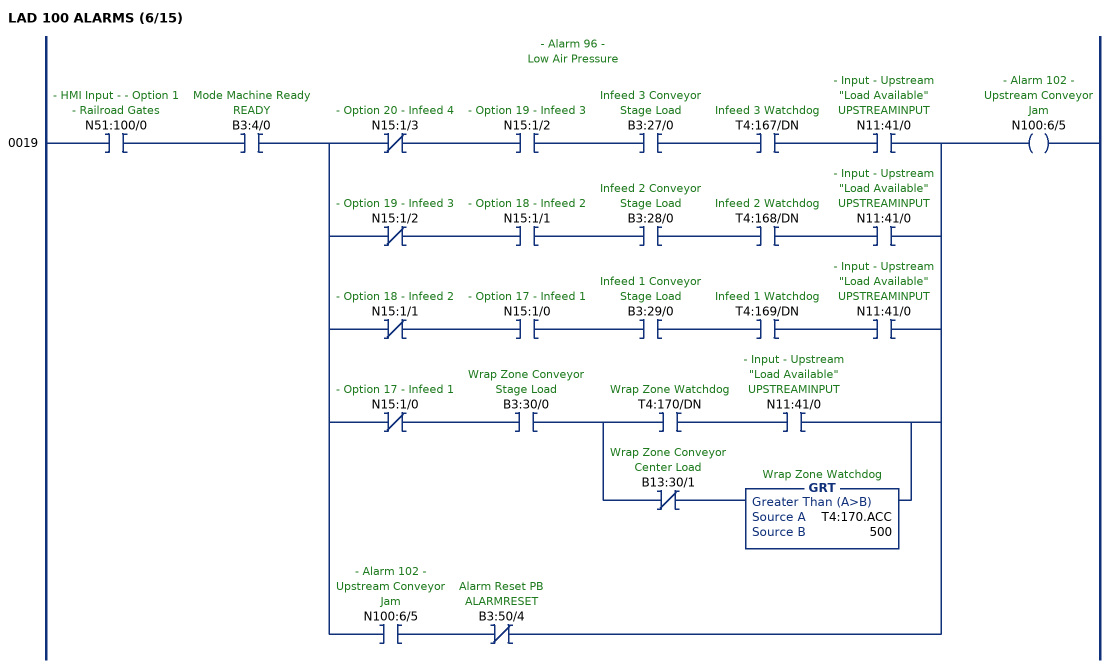
% Rung: 19 %
% - Alarm 96 -
% 
% Low Air Pressure %
SOR XIC N51:100/0 XIC B3:4/0 BST XIO N15:1/3 XIC N15:1/2 XIC B3:27/0 XIC T4:167/DN XIC N11:41/0 NXB XIO N15:1/2 XIC N15:1/1 XIC B3:28/0 XIC T4:168/DN XIC N11:41/0 NXB XIO N15:1/1 XIC N15:1/0 XIC B3:29/0 XIC T4:169/DN XIC N11:41/0 NXB XIO N15:1/0 XIC B3:30/0 BST XIC T4:170/DN XIC N11:41/0 NXB XIO B13:30/1 GRT T4:170.ACC 500 BND NXB XIC N100:6/5 XIO B3:50/4 BND OTE N100:6/5 EOR
%   N51:100/0  "- HMI Input - - Option 1 - Railroad Gates" %
%   B3:4/0  READY  "Mode Machine Ready" %
%   N15:1/3  "- Option 20 - Infeed 4" %
%   N15:1/2  "- Option 19 - Infeed 3" %
%   B3:27/0  "Infeed 3 Conveyor Stage Load" %
%   T4:167  "Infeed 3 Watchdog" %
%   N11:41/0  UPSTREAMINPUT  "- Input - Upstream "Load Available"" %
%   N15:1/1  "- Option 18 - Infeed 2" %
%   B3:28/0  "Infeed 2 Conveyor Stage Load" %
%   T4:168  "Infeed 2 Watchdog" %
%   N15:1/0  "- Option 17 - Infeed 1" %
%   B3:29/0  "Infeed 1 Conveyor Stage Load" %
%   T4:169  "Infeed 1 Watchdog" %
%   B3:30/0  "Wrap Zone Conveyor Stage Load" %
%   T4:170  "Wrap Zone Watchdog" %
%   B13:30/1  "Wrap Zone Conveyor Center Load" %
%   N100:6/5  "- Alarm 102 - Upstream Conveyor Jam" %
%   B3:50/4  ALARMRESET  "Alarm Reset PB" %

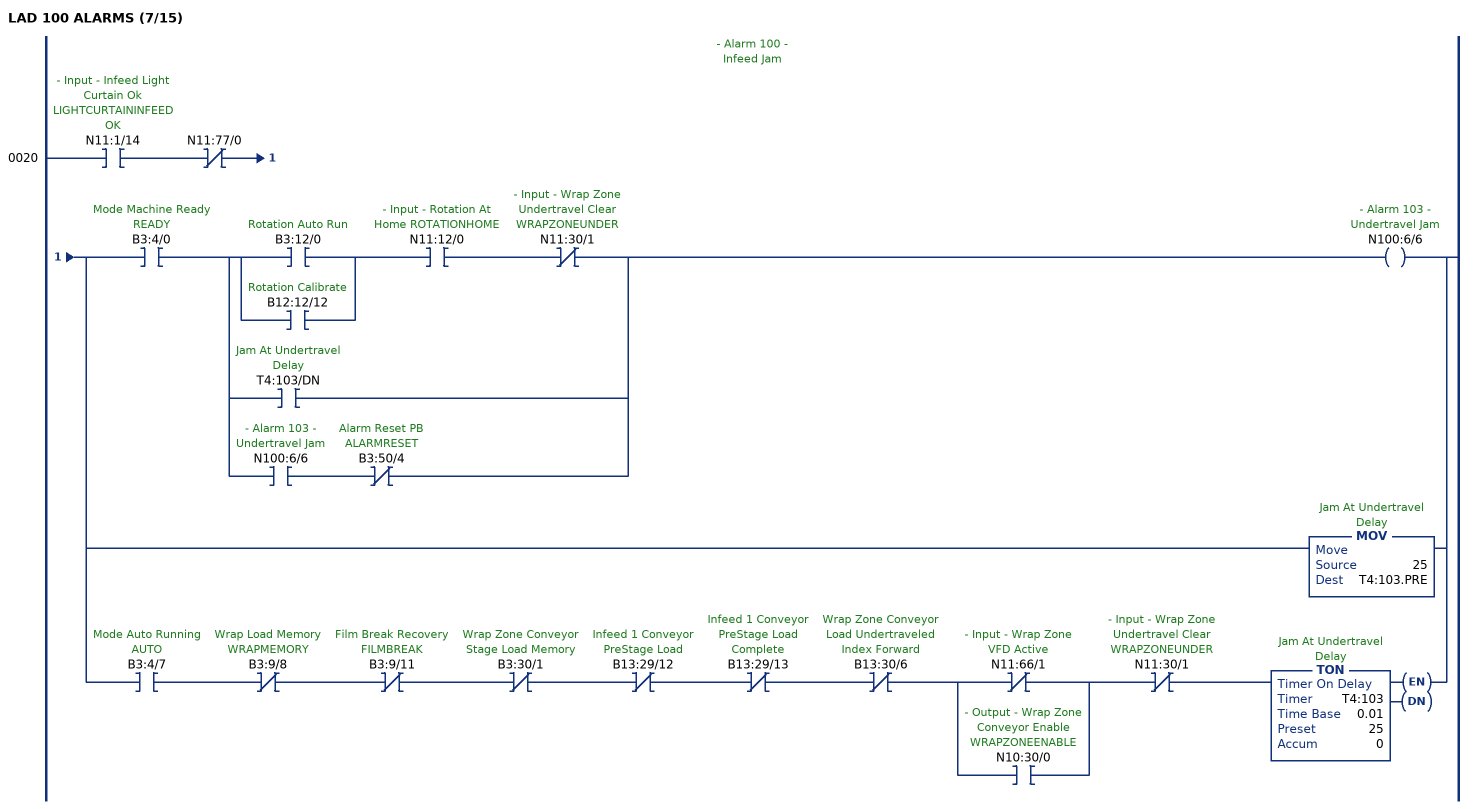
% Rung: 20 %
% - Alarm 100 -
% 
% Infeed Jam %
SOR XIC N11:1/14 XIO N11:77/0 BST XIC B3:4/0 BST BST XIC B3:12/0 NXB XIC B12:12/12 BND XIC N11:12/0 XIO N11:30/1 NXB XIC T4:103/DN NXB XIC N100:6/6 XIO B3:50/4 BND OTE N100:6/6 NXB MOV 25 T4:103.PRE NXB XIC B3:4/7 XIO B3:9/8 XIO B3:9/11 XIO B3:30/1 XIO B13:29/12 XIO B13:29/13 XIO B13:30/6 BST XIO N11:66/1 NXB XIC N10:30/0 BND XIO N11:30/1 TON T4:103 0.01 25 0 BND EOR
%   N11:1/14  LIGHTCURTAININFEEDOK  "- Input - Infeed Light Curtain Ok" %
%   B3:4/0  READY  "Mode Machine Ready" %
%   B3:12/0  "Rotation Auto Run" %
%   B12:12/12  "Rotation Calibrate" %
%   N11:12/0  ROTATIONHOME  "- Input - Rotation At Home" %
%   N11:30/1  WRAPZONEUNDER  "- Input - Wrap Zone Undertravel Clear" %
%   T4:103  "Jam At Undertravel Delay" %
%   N100:6/6  "- Alarm 103 - Undertravel Jam" %
%   B3:50/4  ALARMRESET  "Alarm Reset PB" %
%   B3:4/7  AUTO  "Mode Auto Running" %
%   B3:9/8  WRAPMEMORY  "Wrap Load Memory" %
%   B3:9/11  FILMBREAK  "Film Break Recovery" %
%   B3:30/1  "Wrap Zone Conveyor Stage Load Memory" %
%   B13:29/12  "Infeed 1 Conveyor PreStage Load" %
%   B13:29/13  "Infeed 1 Conveyor PreStage Load Complete" %
%   B13:30/6  "Wrap Zone Conveyor Load Undertraveled Index Forward" %
%   N11:66/1  "- Input - Wrap Zone VFD Active" %
%   N10:30/0  WRAPZONEENABLE  "- Output - Wrap Zone Conveyor Enable" %

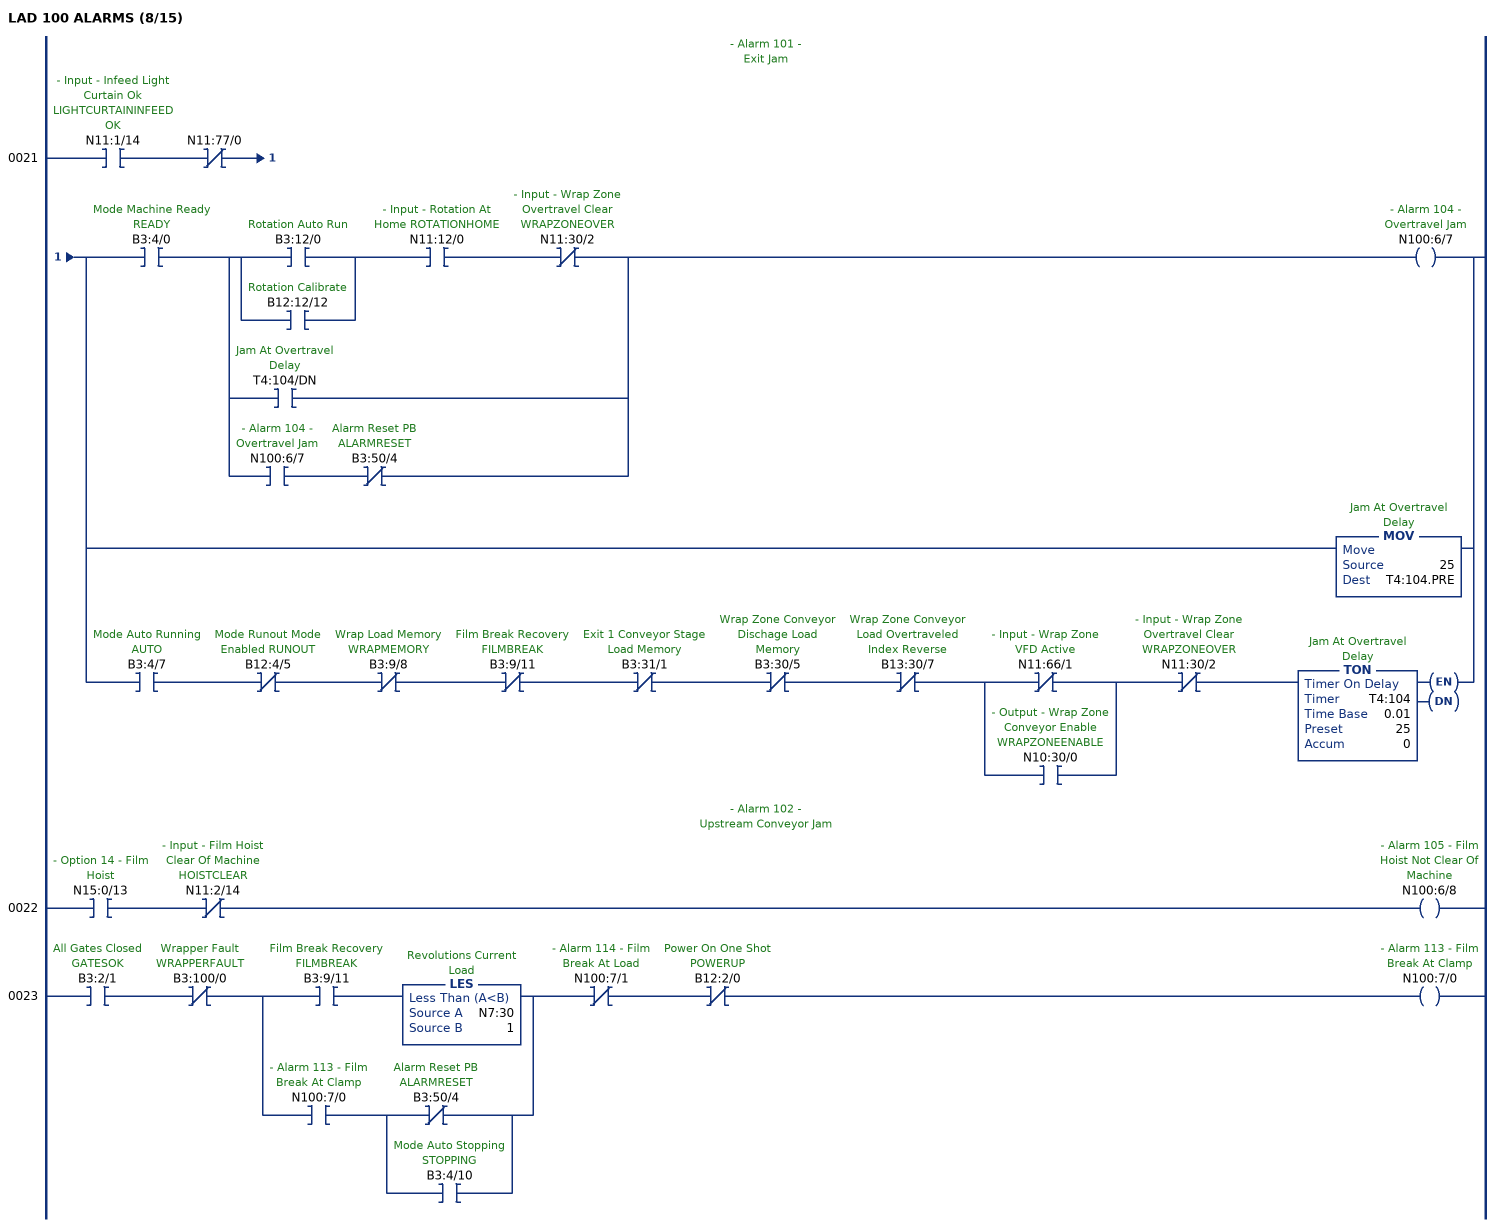
% Rung: 21 %
% - Alarm 101 -
% 
% Exit Jam %
SOR XIC N11:1/14 XIO N11:77/0 BST XIC B3:4/0 BST BST XIC B3:12/0 NXB XIC B12:12/12 BND XIC N11:12/0 XIO N11:30/2 NXB XIC T4:104/DN NXB XIC N100:6/7 XIO B3:50/4 BND OTE N100:6/7 NXB MOV 25 T4:104.PRE NXB XIC B3:4/7 XIO B12:4/5 XIO B3:9/8 XIO B3:9/11 XIO B3:31/1 XIO B3:30/5 XIO B13:30/7 BST XIO N11:66/1 NXB XIC N10:30/0 BND XIO N11:30/2 TON T4:104 0.01 25 0 BND EOR
%   N11:1/14  LIGHTCURTAININFEEDOK  "- Input - Infeed Light Curtain Ok" %
%   B3:4/0  READY  "Mode Machine Ready" %
%   B3:12/0  "Rotation Auto Run" %
%   B12:12/12  "Rotation Calibrate" %
%   N11:12/0  ROTATIONHOME  "- Input - Rotation At Home" %
%   N11:30/2  WRAPZONEOVER  "- Input - Wrap Zone Overtravel Clear" %
%   T4:104  "Jam At Overtravel Delay" %
%   N100:6/7  "- Alarm 104 - Overtravel Jam" %
%   B3:50/4  ALARMRESET  "Alarm Reset PB" %
%   B3:4/7  AUTO  "Mode Auto Running" %
%   B12:4/5  RUNOUT  "Mode Runout Mode Enabled" %
%   B3:9/8  WRAPMEMORY  "Wrap Load Memory" %
%   B3:9/11  FILMBREAK  "Film Break Recovery" %
%   B3:31/1  "Exit 1 Conveyor Stage Load Memory" %
%   B3:30/5  "Wrap Zone Conveyor Dischage Load Memory" %
%   B13:30/7  "Wrap Zone Conveyor Load Overtraveled Index Reverse" %
%   N11:66/1  "- Input - Wrap Zone VFD Active" %
%   N10:30/0  WRAPZONEENABLE  "- Output - Wrap Zone Conveyor Enable" %
% Rung: 22 %
% - Alarm 102 -
% 
% Upstream Conveyor Jam %
SOR XIC N15:0/13 XIO N11:2/14 OTE N100:6/8 EOR
%   N15:0/13  "- Option 14 - Film Hoist" %
%   N11:2/14  HOISTCLEAR  "- Input - Film Hoist Clear Of Machine" %
%   N100:6/8  "- Alarm 105 - Film Hoist Not Clear Of Machine" %
% Rung: 23 %
SOR XIC B3:2/1 XIO B3:100/0 BST XIC B3:9/11 LES N7:30 1 NXB XIC N100:7/0 BST XIO B3:50/4 NXB XIC B3:4/10 BND BND XIO N100:7/1 XIO B12:2/0 OTE N100:7/0 EOR
%   B3:2/1  GATESOK  "All Gates Closed" %
%   B3:100/0  WRAPPERFAULT  "Wrapper Fault" %
%   B3:9/11  FILMBREAK  "Film Break Recovery" %
%   N7:30  "Revolutions Current Load" %
%   N100:7/0  "- Alarm 113 - Film Break At Clamp" %
%   B3:50/4  ALARMRESET  "Alarm Reset PB" %
%   B3:4/10  STOPPING  "Mode Auto Stopping" %
%   N100:7/1  "- Alarm 114 - Film Break At Load" %
%   B12:2/0  POWERUP  "Power On One Shot" %

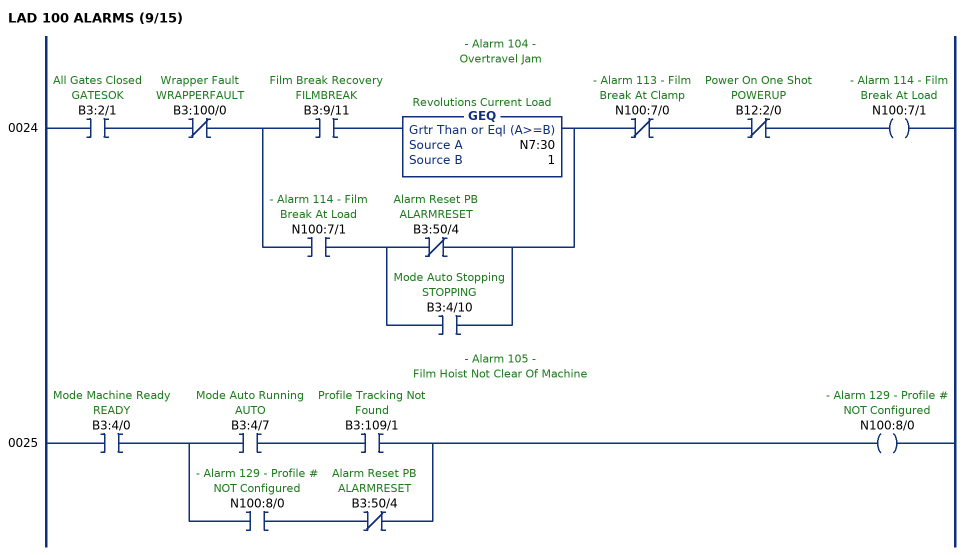
% Rung: 24 %
% - Alarm 104 -
% Overtravel Jam %
SOR XIC B3:2/1 XIO B3:100/0 BST XIC B3:9/11 GEQ N7:30 1 NXB XIC N100:7/1 BST XIO B3:50/4 NXB XIC B3:4/10 BND BND XIO N100:7/0 XIO B12:2/0 OTE N100:7/1 EOR
%   B3:2/1  GATESOK  "All Gates Closed" %
%   B3:100/0  WRAPPERFAULT  "Wrapper Fault" %
%   B3:9/11  FILMBREAK  "Film Break Recovery" %
%   N7:30  "Revolutions Current Load" %
%   N100:7/1  "- Alarm 114 - Film Break At Load" %
%   B3:50/4  ALARMRESET  "Alarm Reset PB" %
%   B3:4/10  STOPPING  "Mode Auto Stopping" %
%   N100:7/0  "- Alarm 113 - Film Break At Clamp" %
%   B12:2/0  POWERUP  "Power On One Shot" %
% Rung: 25 %
% - Alarm 105 -
% 
% Film Hoist Not Clear Of Machine %
SOR XIC B3:4/0 BST XIC B3:4/7 XIC B3:109/1 NXB XIC N100:8/0 XIO B3:50/4 BND OTE N100:8/0 EOR
%   B3:4/0  READY  "Mode Machine Ready" %
%   B3:4/7  AUTO  "Mode Auto Running" %
%   B3:109/1  "Profile Tracking Not Found" %
%   N100:8/0  "- Alarm 129 - Profile # NOT Configured" %
%   B3:50/4  ALARMRESET  "Alarm Reset PB" %

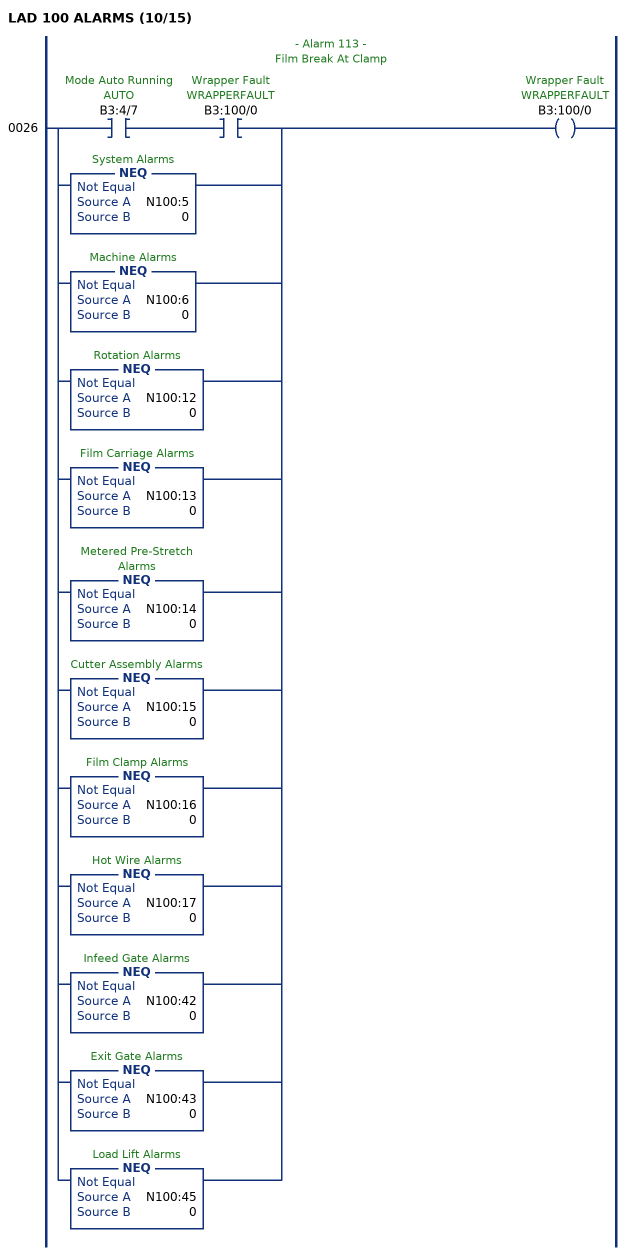
% Rung: 26 %
% - Alarm 113 -
% 
% Film Break At Clamp %
SOR BST XIC B3:4/7 XIC B3:100/0 NXB NEQ N100:5 0 NXB NEQ N100:6 0 NXB NEQ N100:12 0 NXB NEQ N100:13 0 NXB NEQ N100:14 0 NXB NEQ N100:15 0 NXB NEQ N100:16 0 NXB NEQ N100:17 0 NXB NEQ N100:42 0 NXB NEQ N100:43 0 NXB NEQ N100:45 0 BND OTE B3:100/0 EOR
%   B3:4/7  AUTO  "Mode Auto Running" %
%   B3:100/0  WRAPPERFAULT  "Wrapper Fault" %
%   N100:5  "System Alarms" %
%   N100:6  "Machine Alarms" %
%   N100:12  "Rotation Alarms" %
%   N100:13  "Film Carriage Alarms" %
%   N100:14  "Metered Pre-Stretch Alarms" %
%   N100:15  "Cutter Assembly Alarms" %
%   N100:16  "Film Clamp Alarms" %
%   N100:17  "Hot Wire Alarms" %
%   N100:42  "Infeed Gate Alarms" %
%   N100:43  "Exit Gate Alarms" %
%   N100:45  "Load Lift Alarms" %

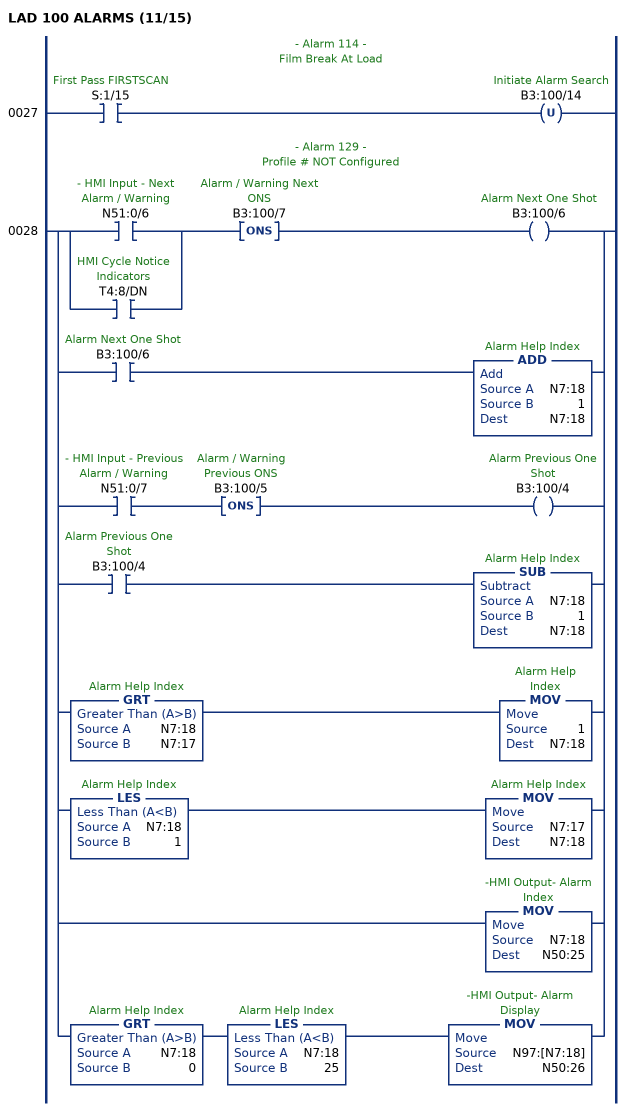
% Rung: 27 %
% - Alarm 114 -
% 
% Film Break At Load %
SOR XIC S:1/15 OTU B3:100/14 EOR
%   S:1/15  FIRSTSCAN  "First Pass" %
%   B3:100/14  "Initiate Alarm Search" %
% Rung: 28 %
% - Alarm 129 -
% 
% Profile # NOT Configured %
SOR BST BST XIC N51:0/6 NXB XIC T4:8/DN BND ONS B3:100/7 OTE B3:100/6 NXB XIC B3:100/6 ADD N7:18 1 N7:18 NXB XIC N51:0/7 ONS B3:100/5 OTE B3:100/4 NXB XIC B3:100/4 SUB N7:18 1 N7:18 NXB GRT N7:18 N7:17 MOV 1 N7:18 NXB LES N7:18 1 MOV N7:17 N7:18 NXB MOV N7:18 N50:25 NXB GRT N7:18 0 LES N7:18 25 MOV N97:[N7:18] N50:26 BND EOR
%   N51:0/6  "- HMI Input - Next Alarm / Warning" %
%   T4:8  "HMI Cycle Notice Indicators" %
%   B3:100/7  "Alarm / Warning Next ONS" %
%   B3:100/6  "Alarm Next One Shot" %
%   N7:18  "Alarm Help Index" %
%   N51:0/7  "- HMI Input - Previous Alarm / Warning" %
%   B3:100/5  "Alarm / Warning Previous ONS" %
%   B3:100/4  "Alarm Previous One Shot" %
%   N7:17  ALARMCOUNT  "Alarm Count" %
%   N50:25  "-HMI Output- Alarm Index" %
%   N50:26  "-HMI Output- Alarm Display" %

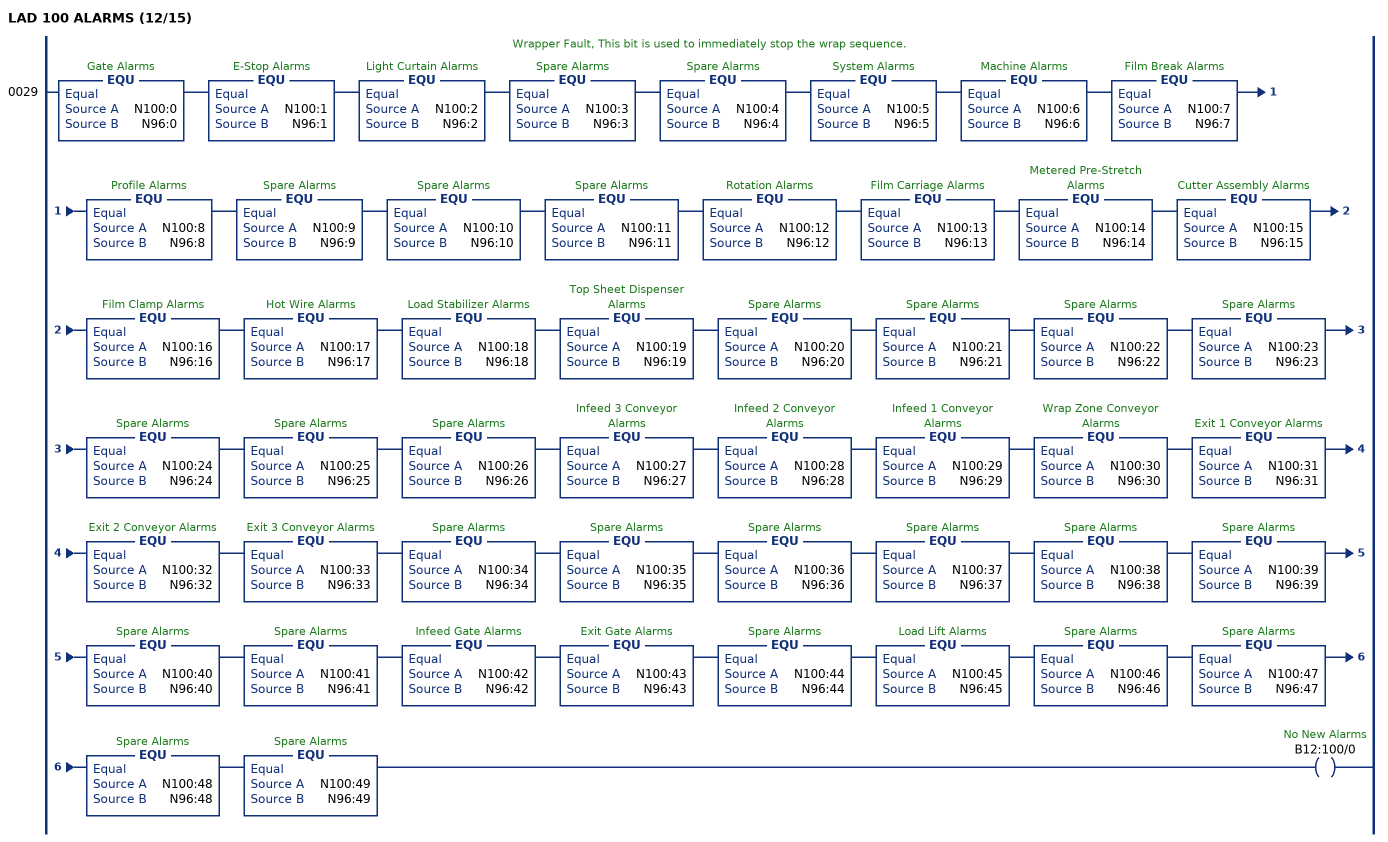
% Rung: 29 %
% Wrapper Fault, This bit is used to immediately stop the wrap sequence. %
SOR EQU N100:0 N96:0 EQU N100:1 N96:1 EQU N100:2 N96:2 EQU N100:3 N96:3 EQU N100:4 N96:4 EQU N100:5 N96:5 EQU N100:6 N96:6 EQU N100:7 N96:7 EQU N100:8 N96:8 EQU N100:9 N96:9 EQU N100:10 N96:10 EQU N100:11 N96:11 EQU N100:12 N96:12 EQU N100:13 N96:13 EQU N100:14 N96:14 EQU N100:15 N96:15 EQU N100:16 N96:16 EQU N100:17 N96:17 EQU N100:18 N96:18 EQU N100:19 N96:19 EQU N100:20 N96:20 EQU N100:21 N96:21 EQU N100:22 N96:22 EQU N100:23 N96:23 EQU N100:24 N96:24 EQU N100:25 N96:25 EQU N100:26 N96:26 EQU N100:27 N96:27 EQU N100:28 N96:28 EQU N100:29 N96:29 EQU N100:30 N96:30 EQU N100:31 N96:31 EQU N100:32 N96:32 EQU N100:33 N96:33 EQU N100:34 N96:34 EQU N100:35 N96:35 EQU N100:36 N96:36 EQU N100:37 N96:37 EQU N100:38 N96:38 EQU N100:39 N96:39 EQU N100:40 N96:40 EQU N100:41 N96:41 EQU N100:42 N96:42 EQU N100:43 N96:43 EQU N100:44 N96:44 EQU N100:45 N96:45 EQU N100:46 N96:46 EQU N100:47 N96:47 EQU N100:48 N96:48 EQU N100:49 N96:49 OTE B12:100/0 EOR
%   N100:0  "Gate Alarms" %
%   N96:0  "ALARM ARRAY COMPARISON" %
%   N100:1  "E-Stop Alarms" %
%   N100:2  "Light Curtain Alarms" %
%   N100:3  "Spare Alarms" %
%   N100:4  "Spare Alarms" %
%   N100:5  "System Alarms" %
%   N100:6  "Machine Alarms" %
%   N100:7  "Film Break Alarms" %
%   N100:8  "Profile Alarms" %
%   N100:9  "Spare Alarms" %
%   N100:10  "Spare Alarms" %
%   N100:11  "Spare Alarms" %
%   N100:12  "Rotation Alarms" %
%   N100:13  "Film Carriage Alarms" %
%   N100:14  "Metered Pre-Stretch Alarms" %
%   N100:15  "Cutter Assembly Alarms" %
%   N100:16  "Film Clamp Alarms" %
%   N100:17  "Hot Wire Alarms" %
%   N100:18  "Load Stabilizer Alarms" %
%   N100:19  "Top Sheet Dispenser Alarms" %
%   N100:20  "Spare Alarms" %
%   N100:21  "Spare Alarms" %
%   N100:22  "Spare Alarms" %
%   N100:23  "Spare Alarms" %
%   N100:24  "Spare Alarms" %
%   N100:25  "Spare Alarms" %
%   N100:26  "Spare Alarms" %
%   N100:27  "Infeed 3 Conveyor Alarms" %
%   N100:28  "Infeed 2 Conveyor Alarms" %
%   N100:29  "Infeed 1 Conveyor Alarms" %
%   N100:30  "Wrap Zone Conveyor Alarms" %
%   N100:31  "Exit 1 Conveyor Alarms" %
%   N100:32  "Exit 2 Conveyor Alarms" %
%   N100:33  "Exit 3 Conveyor Alarms" %
%   N100:34  "Spare Alarms" %
%   N100:35  "Spare Alarms" %
%   N100:36  "Spare Alarms" %
%   N100:37  "Spare Alarms" %
%   N100:38  "Spare Alarms" %
%   N100:39  "Spare Alarms" %
%   N100:40  "Spare Alarms" %
%   N100:41  "Spare Alarms" %
%   N100:42  "Infeed Gate Alarms" %
%   N100:43  "Exit Gate Alarms" %
%   N100:44  "Spare Alarms" %
%   N100:45  "Load Lift Alarms" %
%   N100:46  "Spare Alarms" %
%   N100:47  "Spare Alarms" %
%   N100:48  "Spare Alarms" %
%   N100:49  "Spare Alarms" %
%   B12:100/0  "No New Alarms" %

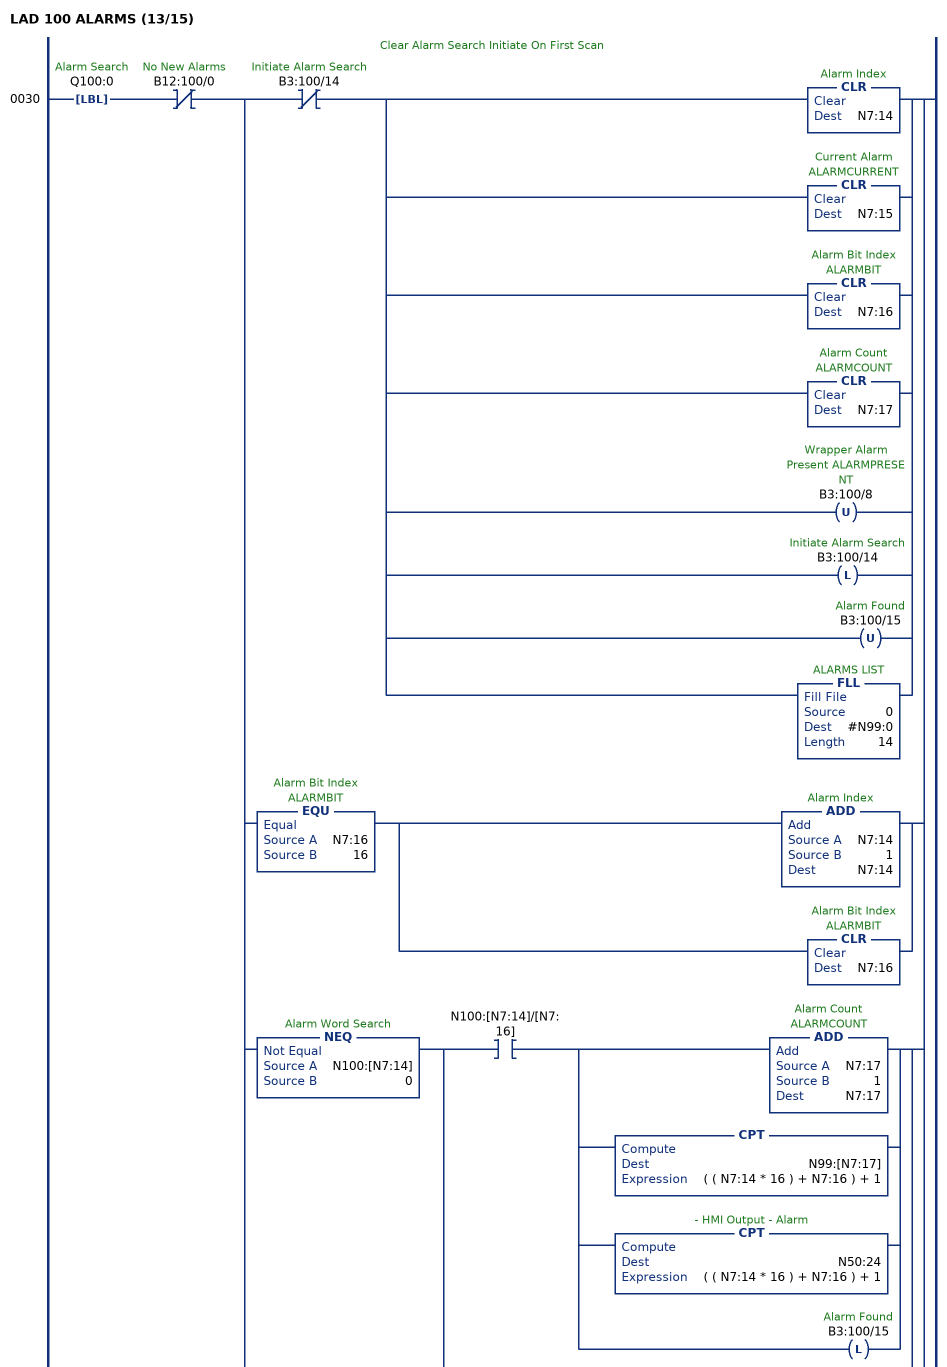

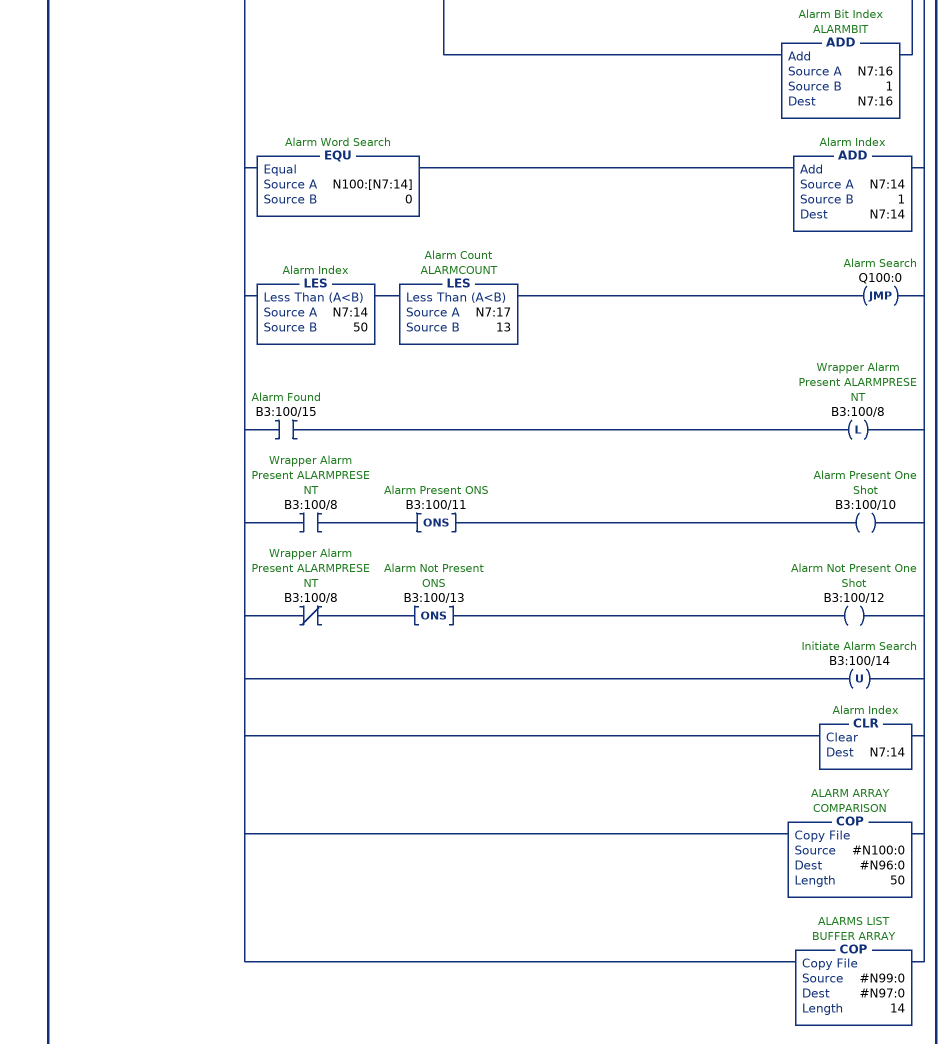
% Rung: 30 %
% Clear Alarm Search Initiate On First Scan %
SOR LBL Q100:0 XIO B12:100/0 BST XIO B3:100/14 BST CLR N7:14 NXB CLR N7:15 NXB CLR N7:16 NXB CLR N7:17 NXB OTU B3:100/8 NXB OTL B3:100/14 NXB OTU B3:100/15 NXB FLL 0 #N99:0 14 BND NXB EQU N7:16 16 BST ADD N7:14 1 N7:14 NXB CLR N7:16 BND NXB NEQ N100:[N7:14] 0 BST XIC N100:[N7:14]/[N7:16] BST ADD N7:17 1 N7:17 NXB CPT N99:[N7:17] " ( ( N7:14 * 16 ) + N7:16 ) + 1 " NXB CPT N50:24 " ( ( N7:14 * 16 ) + N7:16 ) + 1 " NXB OTL B3:100/15 BND NXB ADD N7:16 1 N7:16 BND NXB EQU N100:[N7:14] 0 ADD N7:14 1 N7:14 NXB LES N7:14 50 LES N7:17 13 JMP Q100:0 NXB XIC B3:100/15 OTL B3:100/8 NXB XIC B3:100/8 ONS B3:100/11 OTE B3:100/10 NXB XIO B3:100/8 ONS B3:100/13 OTE B3:100/12 NXB OTU B3:100/14 NXB CLR N7:14 NXB COP #N100:0 #N96:0 50 NXB COP #N99:0 #N97:0 14 BND EOR
%   Q100:0  "Alarm Search" %
%   B12:100/0  "No New Alarms" %
%   B3:100/14  "Initiate Alarm Search" %
%   N7:14  "Alarm Index" %
%   N7:15  ALARMCURRENT  "Current Alarm" %
%   N7:16  ALARMBIT  "Alarm Bit Index" %
%   N7:17  ALARMCOUNT  "Alarm Count" %
%   B3:100/8  ALARMPRESENT  "Wrapper Alarm Present" %
%   B3:100/15  "Alarm Found" %
%   N99:0  "ALARMS LIST" %
%   N100:[N7:14]  "Alarm Word Search" %
%   N50:24  "- HMI Output - Alarm" %
%   B3:100/11  "Alarm Present ONS" %
%   B3:100/10  "Alarm Present One Shot" %
%   B3:100/13  "Alarm Not Present ONS" %
%   B3:100/12  "Alarm Not Present One Shot" %
%   N100:0  "Gate Alarms" %
%   N96:0  "ALARM ARRAY COMPARISON" %
%   N97:0  "ALARMS LIST BUFFER ARRAY" %

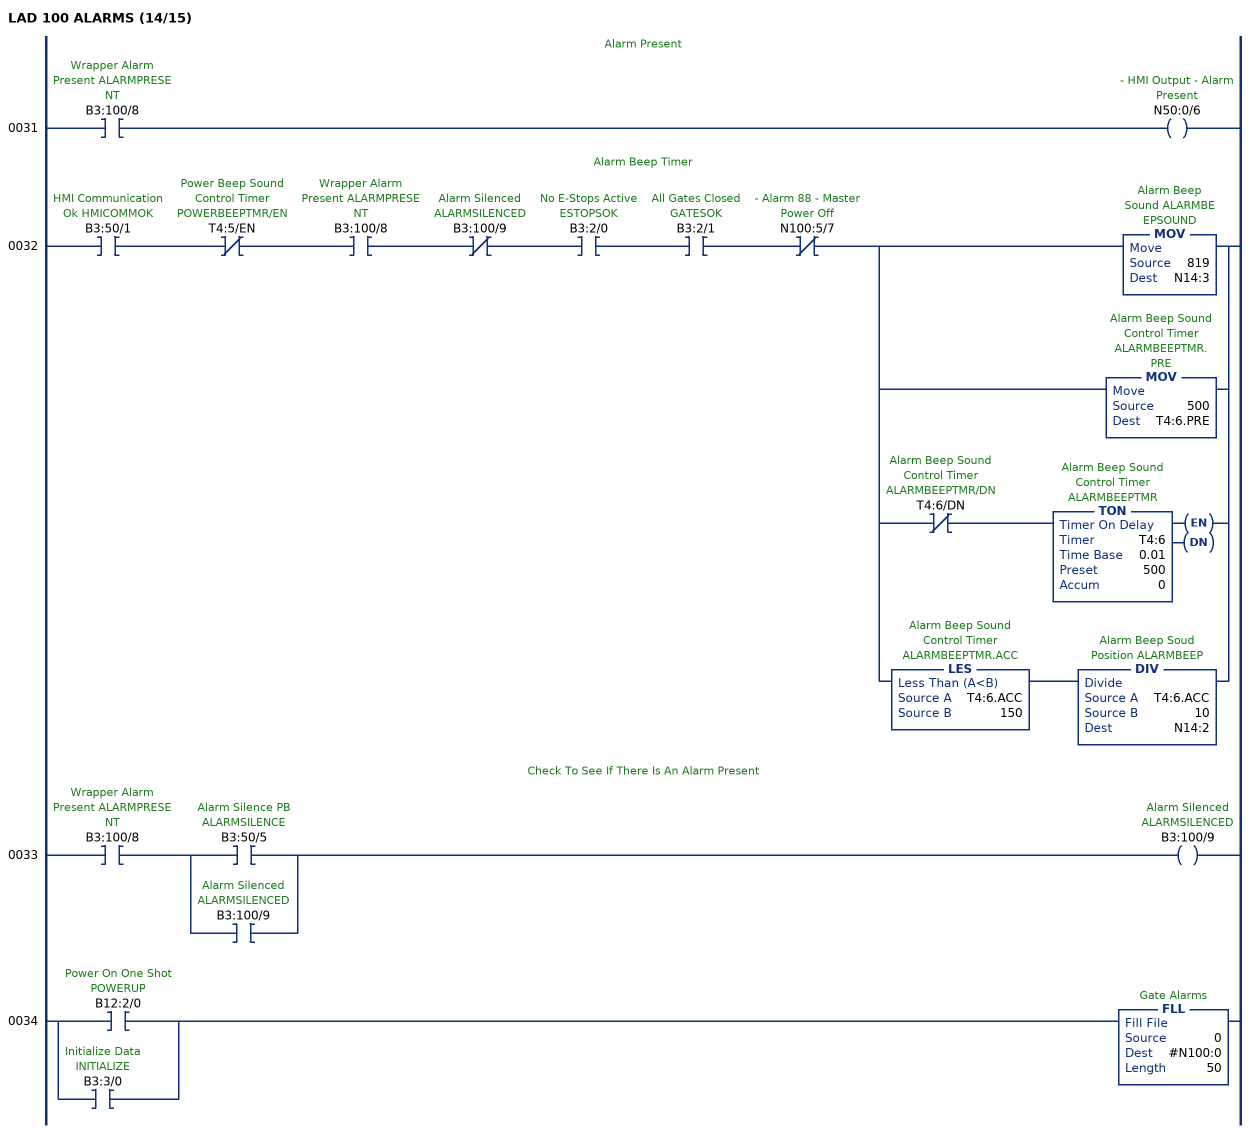
% Rung: 31 %
% Alarm Present %
SOR XIC B3:100/8 OTE N50:0/6 EOR
%   B3:100/8  ALARMPRESENT  "Wrapper Alarm Present" %
%   N50:0/6  "- HMI Output - Alarm Present" %
% Rung: 32 %
% Alarm Beep Timer %
SOR XIC B3:50/1 XIO T4:5/EN XIC B3:100/8 XIO B3:100/9 XIC B3:2/0 XIC B3:2/1 XIO N100:5/7 BST MOV 819 N14:3 NXB MOV 500 T4:6.PRE NXB XIO T4:6/DN TON T4:6 0.01 500 0 NXB LES T4:6.ACC 150 DIV T4:6.ACC 10 N14:2 BND EOR
%   B3:50/1  HMICOMMOK  "HMI Communication Ok" %
%   T4:5  POWERBEEPTMR  "Power Beep Sound Control Timer" %
%   B3:100/8  ALARMPRESENT  "Wrapper Alarm Present" %
%   B3:100/9  ALARMSILENCED  "Alarm Silenced" %
%   B3:2/0  ESTOPSOK  "No E-Stops Active" %
%   B3:2/1  GATESOK  "All Gates Closed" %
%   N100:5/7  "- Alarm 88 - Master Power Off" %
%   N14:3  ALARMBEEPSOUND  "Alarm Beep Sound" %
%   T4:6  ALARMBEEPTMR  "Alarm Beep Sound Control Timer" %
%   N14:2  ALARMBEEP  "Alarm Beep Soud Position" %
% Rung: 33 %
% Check To See If There Is An Alarm Present %
SOR XIC B3:100/8 BST XIC B3:50/5 NXB XIC B3:100/9 BND OTE B3:100/9 EOR
%   B3:100/8  ALARMPRESENT  "Wrapper Alarm Present" %
%   B3:50/5  ALARMSILENCE  "Alarm Silence PB" %
%   B3:100/9  ALARMSILENCED  "Alarm Silenced" %
% Rung: 34 %
SOR BST XIC B12:2/0 NXB XIC B3:3/0 BND FLL 0 #N100:0 50 EOR
%   B12:2/0  POWERUP  "Power On One Shot" %
%   B3:3/0  INITIALIZE  "Initialize Data" %
%   N100:0  "Gate Alarms" %

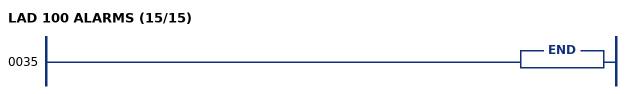
% Rung: 35 %
SOR END EOR

LADDER 101 "MAINT"
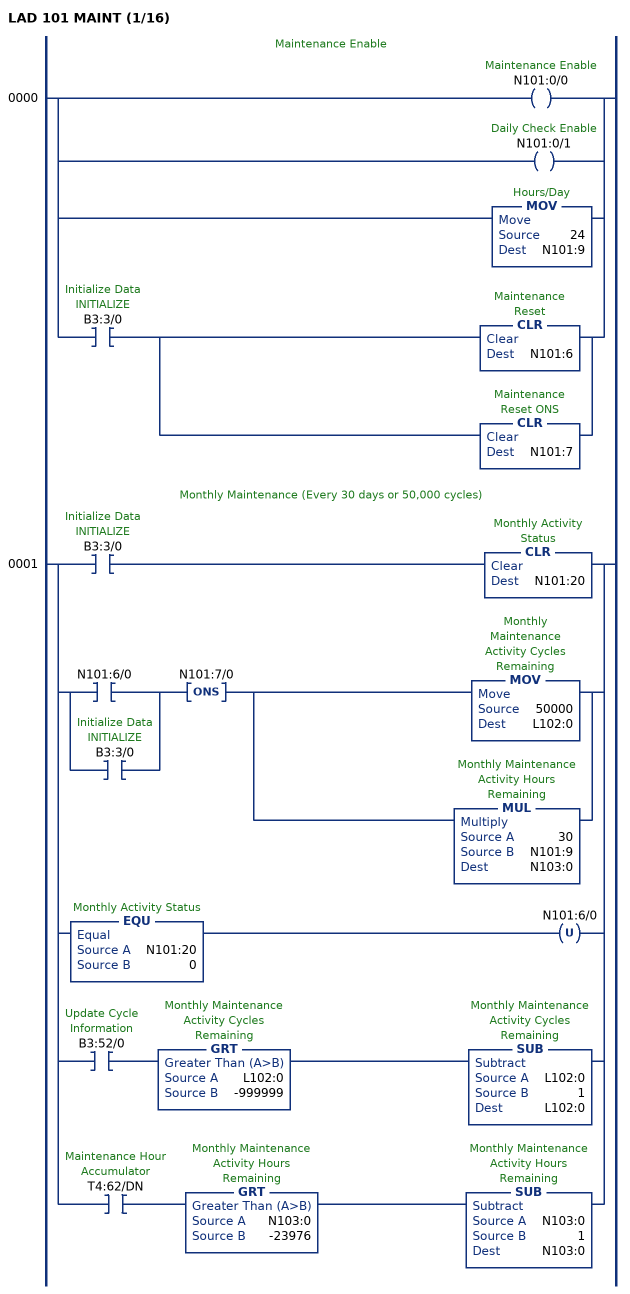
% Rung: 0 %
% Maintenance Enable %
SOR BST OTE N101:0/0 NXB OTE N101:0/1 NXB MOV 24 N101:9 NXB XIC B3:3/0 BST CLR N101:6 NXB CLR N101:7 BND BND EOR
%   N101:0/0  "Maintenance Enable" %
%   N101:0/1  "Daily Check Enable" %
%   N101:9  "Hours/Day" %
%   B3:3/0  INITIALIZE  "Initialize Data" %
%   N101:6  "Maintenance Reset" %
%   N101:7  "Maintenance Reset ONS" %
% Rung: 1 %
% Monthly Maintenance (Every 30 days or 50,000 cycles) %
SOR BST XIC B3:3/0 CLR N101:20 NXB BST XIC N101:6/0 NXB XIC B3:3/0 BND ONS N101:7/0 BST MOV 50000 L102:0 NXB MUL 30 N101:9 N103:0 BND NXB EQU N101:20 0 OTU N101:6/0 NXB XIC B3:52/0 GRT L102:0 -999999 SUB L102:0 1 L102:0 NXB XIC T4:62/DN GRT N103:0 -23976 SUB N103:0 1 N103:0 BND EOR
%   B3:3/0  INITIALIZE  "Initialize Data" %
%   N101:20  "Monthly Activity Status" %
%   L102:0  "Monthly Maintenance Activity Cycles Remaining" %
%   N101:9  "Hours/Day" %
%   N103:0  "Monthly Maintenance Activity Hours Remaining" %
%   B3:52/0  "Update Cycle Information" %
%   T4:62  "Maintenance Hour Accumulator" %

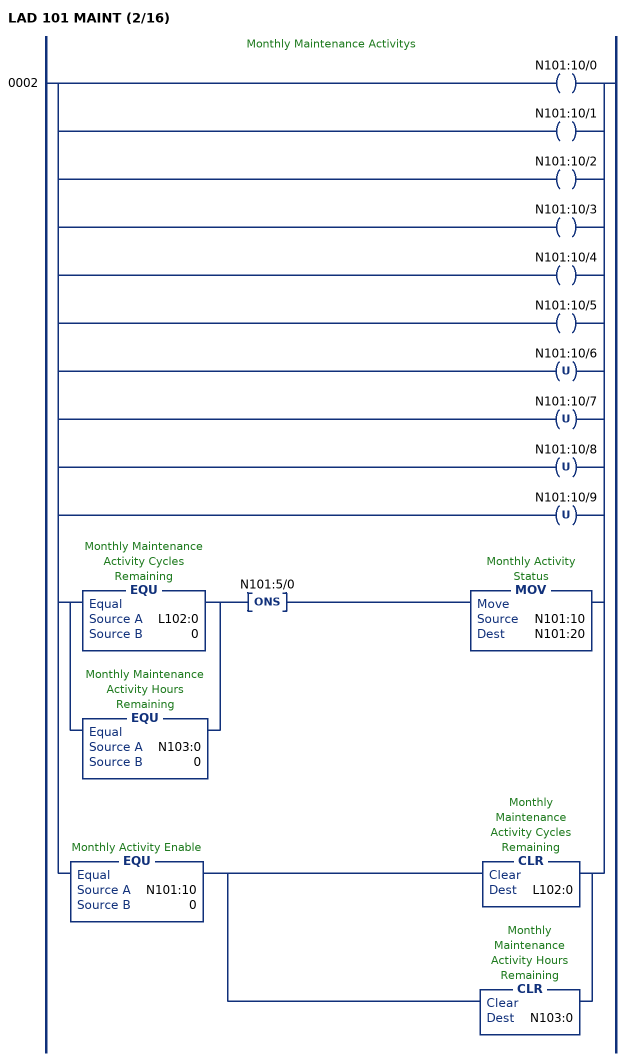
% Rung: 2 %
% Monthly Maintenance Activitys %
SOR BST OTE N101:10/0 NXB OTE N101:10/1 NXB OTE N101:10/2 NXB OTE N101:10/3 NXB OTE N101:10/4 NXB OTE N101:10/5 NXB OTU N101:10/6 NXB OTU N101:10/7 NXB OTU N101:10/8 NXB OTU N101:10/9 NXB BST EQU L102:0 0 NXB EQU N103:0 0 BND ONS N101:5/0 MOV N101:10 N101:20 NXB EQU N101:10 0 BST CLR L102:0 NXB CLR N103:0 BND BND EOR
%   L102:0  "Monthly Maintenance Activity Cycles Remaining" %
%   N103:0  "Monthly Maintenance Activity Hours Remaining" %
%   N101:10  "Monthly Activity Enable" %
%   N101:20  "Monthly Activity Status" %

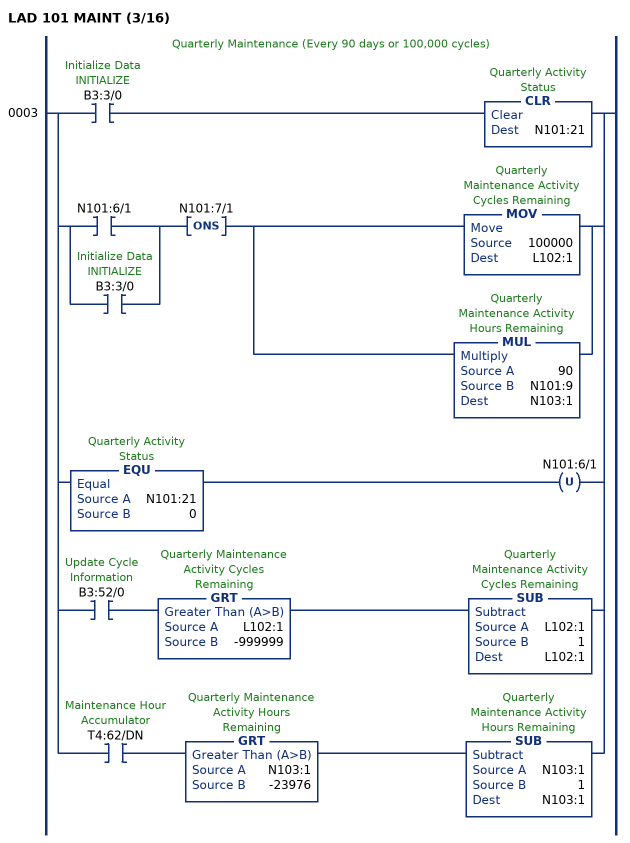
% Rung: 3 %
% Quarterly Maintenance (Every 90 days or 100,000 cycles) %
SOR BST XIC B3:3/0 CLR N101:21 NXB BST XIC N101:6/1 NXB XIC B3:3/0 BND ONS N101:7/1 BST MOV 100000 L102:1 NXB MUL 90 N101:9 N103:1 BND NXB EQU N101:21 0 OTU N101:6/1 NXB XIC B3:52/0 GRT L102:1 -999999 SUB L102:1 1 L102:1 NXB XIC T4:62/DN GRT N103:1 -23976 SUB N103:1 1 N103:1 BND EOR
%   B3:3/0  INITIALIZE  "Initialize Data" %
%   N101:21  "Quarterly Activity Status" %
%   L102:1  "Quarterly Maintenance Activity Cycles Remaining" %
%   N101:9  "Hours/Day" %
%   N103:1  "Quarterly Maintenance Activity Hours Remaining" %
%   B3:52/0  "Update Cycle Information" %
%   T4:62  "Maintenance Hour Accumulator" %

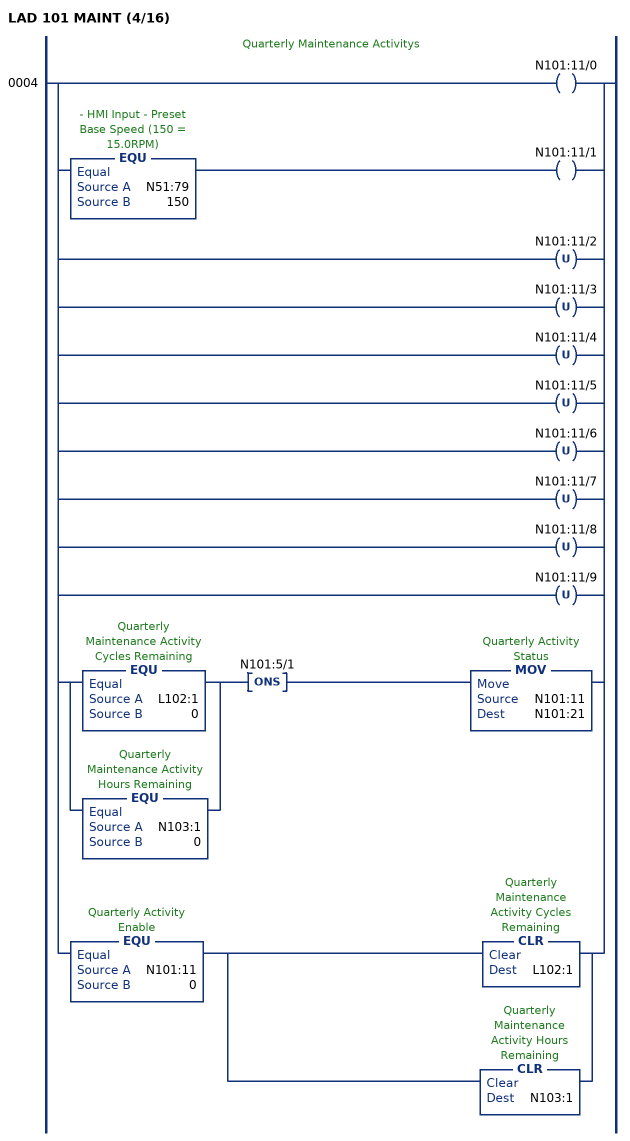
% Rung: 4 %
% Quarterly Maintenance Activitys %
SOR BST OTE N101:11/0 NXB EQU N51:79 150 OTE N101:11/1 NXB OTU N101:11/2 NXB OTU N101:11/3 NXB OTU N101:11/4 NXB OTU N101:11/5 NXB OTU N101:11/6 NXB OTU N101:11/7 NXB OTU N101:11/8 NXB OTU N101:11/9 NXB BST EQU L102:1 0 NXB EQU N103:1 0 BND ONS N101:5/1 MOV N101:11 N101:21 NXB EQU N101:11 0 BST CLR L102:1 NXB CLR N103:1 BND BND EOR
%   N51:79  "- HMI Input - Preset Base Speed (150 = 15.0RPM)" %
%   L102:1  "Quarterly Maintenance Activity Cycles Remaining" %
%   N103:1  "Quarterly Maintenance Activity Hours Remaining" %
%   N101:11  "Quarterly Activity Enable" %
%   N101:21  "Quarterly Activity Status" %

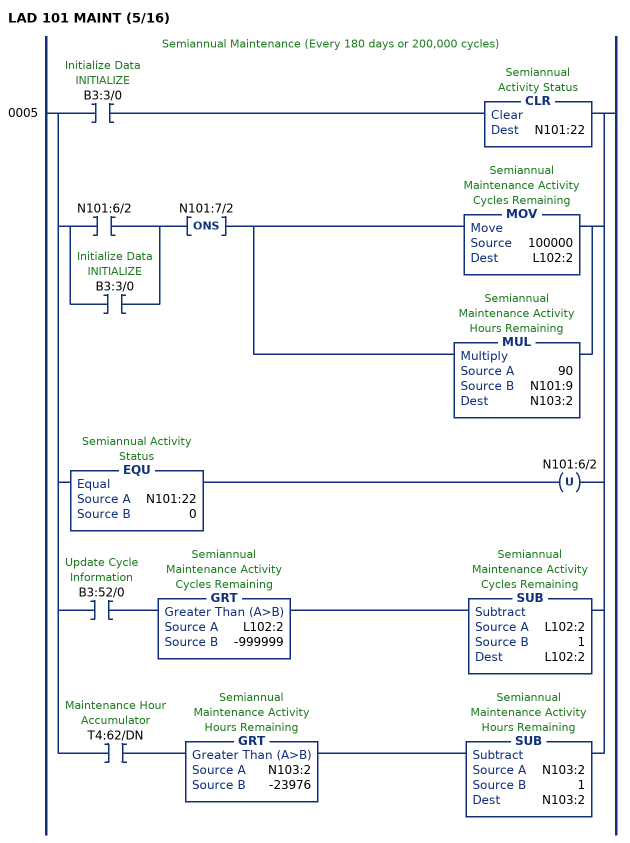
% Rung: 5 %
% Semiannual Maintenance (Every 180 days or 200,000 cycles) %
SOR BST XIC B3:3/0 CLR N101:22 NXB BST XIC N101:6/2 NXB XIC B3:3/0 BND ONS N101:7/2 BST MOV 100000 L102:2 NXB MUL 90 N101:9 N103:2 BND NXB EQU N101:22 0 OTU N101:6/2 NXB XIC B3:52/0 GRT L102:2 -999999 SUB L102:2 1 L102:2 NXB XIC T4:62/DN GRT N103:2 -23976 SUB N103:2 1 N103:2 BND EOR
%   B3:3/0  INITIALIZE  "Initialize Data" %
%   N101:22  "Semiannual Activity Status" %
%   L102:2  "Semiannual Maintenance Activity Cycles Remaining" %
%   N101:9  "Hours/Day" %
%   N103:2  "Semiannual Maintenance Activity Hours Remaining" %
%   B3:52/0  "Update Cycle Information" %
%   T4:62  "Maintenance Hour Accumulator" %

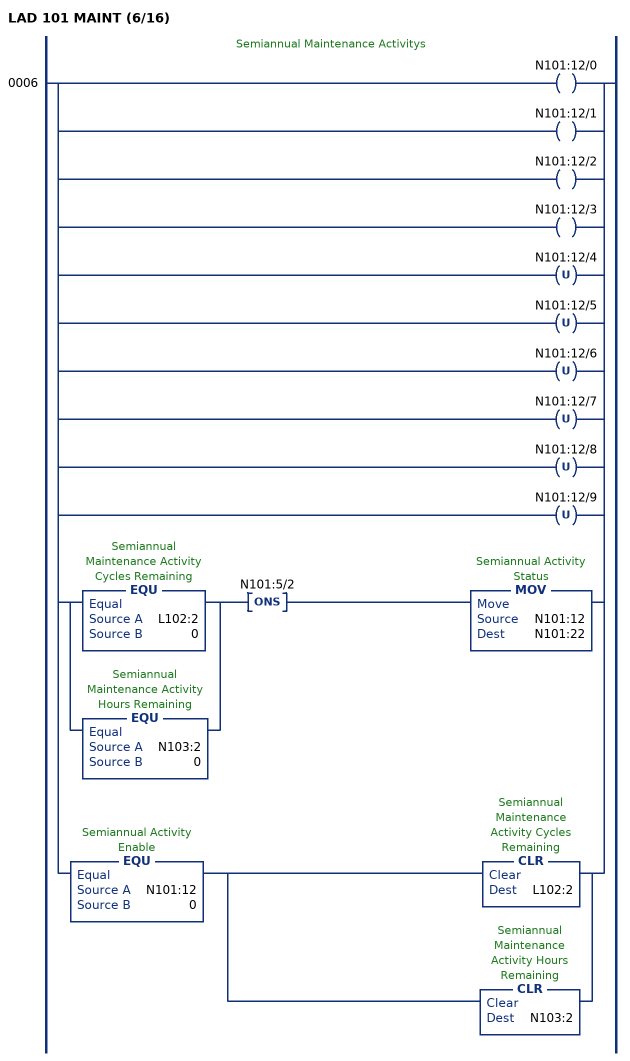
% Rung: 6 %
% Semiannual Maintenance Activitys %
SOR BST OTE N101:12/0 NXB OTE N101:12/1 NXB OTE N101:12/2 NXB OTE N101:12/3 NXB OTU N101:12/4 NXB OTU N101:12/5 NXB OTU N101:12/6 NXB OTU N101:12/7 NXB OTU N101:12/8 NXB OTU N101:12/9 NXB BST EQU L102:2 0 NXB EQU N103:2 0 BND ONS N101:5/2 MOV N101:12 N101:22 NXB EQU N101:12 0 BST CLR L102:2 NXB CLR N103:2 BND BND EOR
%   L102:2  "Semiannual Maintenance Activity Cycles Remaining" %
%   N103:2  "Semiannual Maintenance Activity Hours Remaining" %
%   N101:12  "Semiannual Activity Enable" %
%   N101:22  "Semiannual Activity Status" %

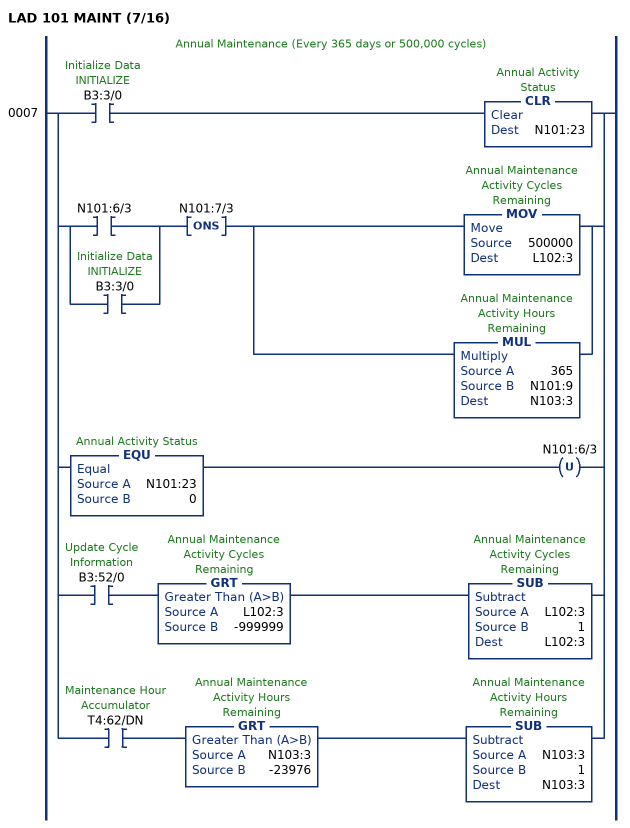
% Rung: 7 %
% Annual Maintenance (Every 365 days or 500,000 cycles) %
SOR BST XIC B3:3/0 CLR N101:23 NXB BST XIC N101:6/3 NXB XIC B3:3/0 BND ONS N101:7/3 BST MOV 500000 L102:3 NXB MUL 365 N101:9 N103:3 BND NXB EQU N101:23 0 OTU N101:6/3 NXB XIC B3:52/0 GRT L102:3 -999999 SUB L102:3 1 L102:3 NXB XIC T4:62/DN GRT N103:3 -23976 SUB N103:3 1 N103:3 BND EOR
%   B3:3/0  INITIALIZE  "Initialize Data" %
%   N101:23  "Annual Activity Status" %
%   L102:3  "Annual Maintenance Activity Cycles Remaining" %
%   N101:9  "Hours/Day" %
%   N103:3  "Annual Maintenance Activity Hours Remaining" %
%   B3:52/0  "Update Cycle Information" %
%   T4:62  "Maintenance Hour Accumulator" %

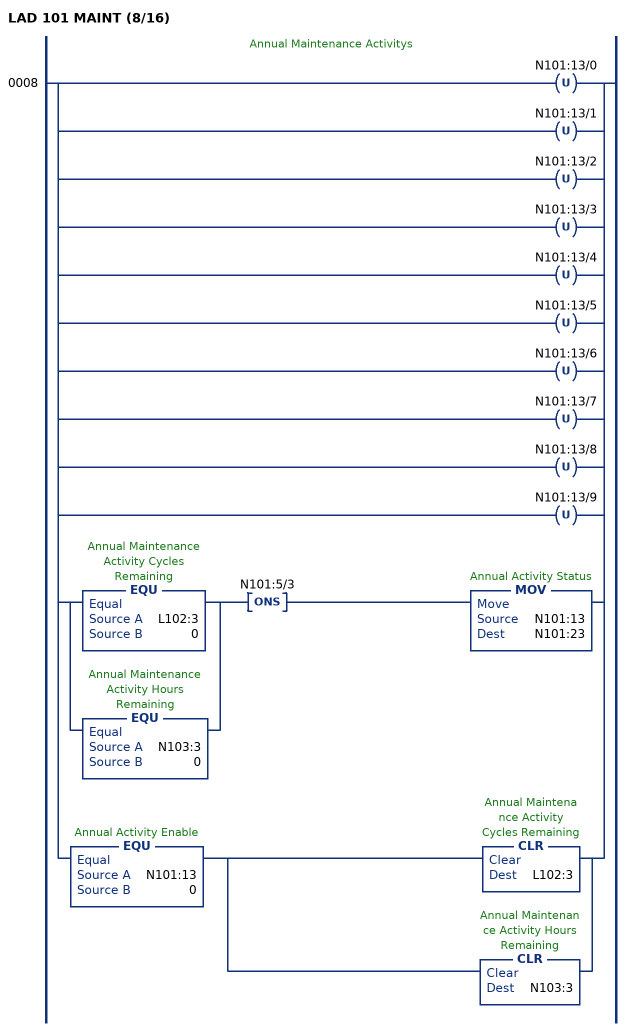
% Rung: 8 %
% Annual Maintenance Activitys %
SOR BST OTU N101:13/0 NXB OTU N101:13/1 NXB OTU N101:13/2 NXB OTU N101:13/3 NXB OTU N101:13/4 NXB OTU N101:13/5 NXB OTU N101:13/6 NXB OTU N101:13/7 NXB OTU N101:13/8 NXB OTU N101:13/9 NXB BST EQU L102:3 0 NXB EQU N103:3 0 BND ONS N101:5/3 MOV N101:13 N101:23 NXB EQU N101:13 0 BST CLR L102:3 NXB CLR N103:3 BND BND EOR
%   L102:3  "Annual Maintenance Activity Cycles Remaining" %
%   N103:3  "Annual Maintenance Activity Hours Remaining" %
%   N101:13  "Annual Activity Enable" %
%   N101:23  "Annual Activity Status" %

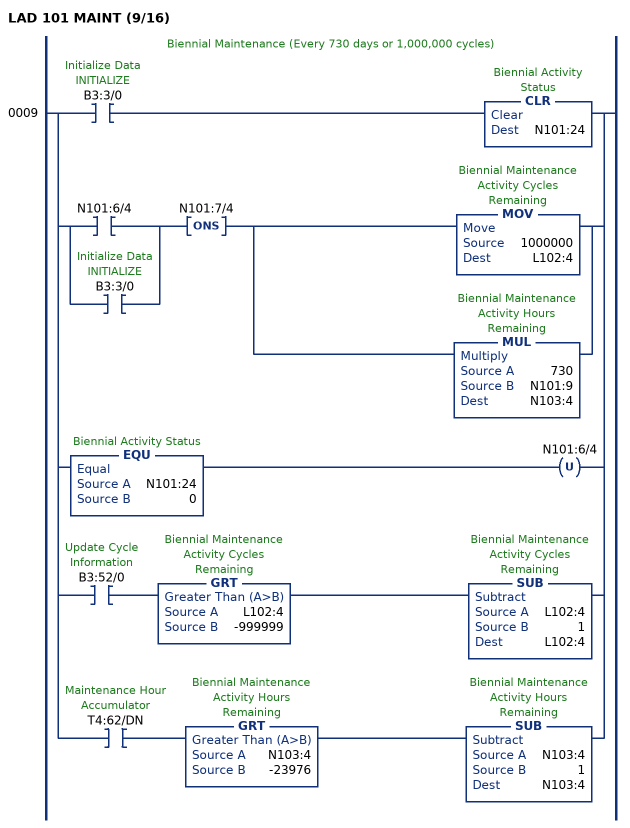
% Rung: 9 %
% Biennial Maintenance (Every 730 days or 1,000,000 cycles) %
SOR BST XIC B3:3/0 CLR N101:24 NXB BST XIC N101:6/4 NXB XIC B3:3/0 BND ONS N101:7/4 BST MOV 1000000 L102:4 NXB MUL 730 N101:9 N103:4 BND NXB EQU N101:24 0 OTU N101:6/4 NXB XIC B3:52/0 GRT L102:4 -999999 SUB L102:4 1 L102:4 NXB XIC T4:62/DN GRT N103:4 -23976 SUB N103:4 1 N103:4 BND EOR
%   B3:3/0  INITIALIZE  "Initialize Data" %
%   N101:24  "Biennial Activity Status" %
%   L102:4  "Biennial Maintenance Activity Cycles Remaining" %
%   N101:9  "Hours/Day" %
%   N103:4  "Biennial Maintenance Activity Hours Remaining" %
%   B3:52/0  "Update Cycle Information" %
%   T4:62  "Maintenance Hour Accumulator" %

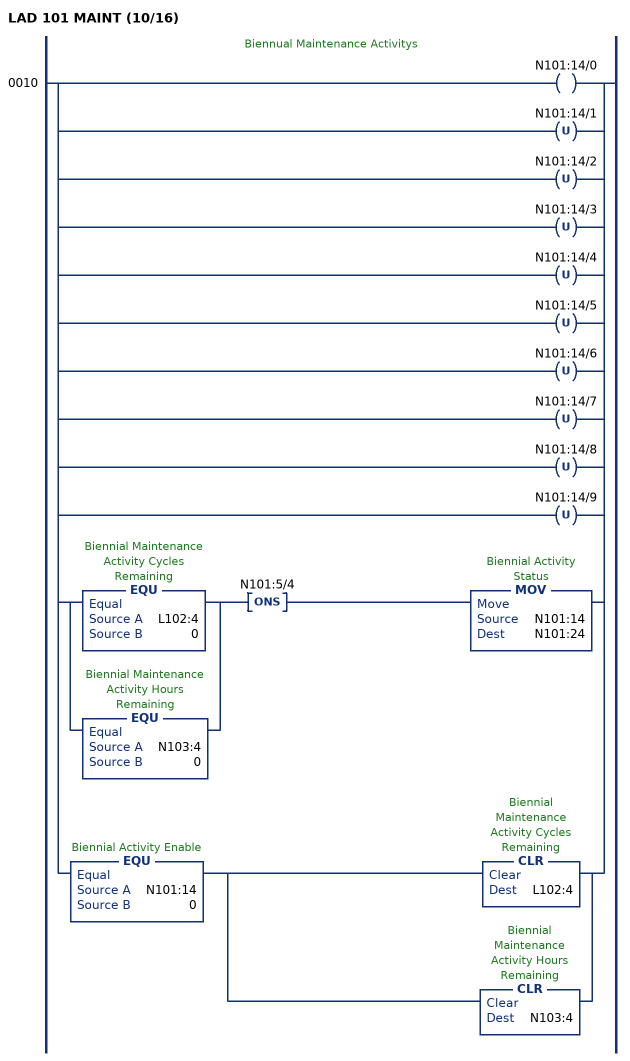
% Rung: 10 %
% Biennual Maintenance Activitys %
SOR BST OTE N101:14/0 NXB OTU N101:14/1 NXB OTU N101:14/2 NXB OTU N101:14/3 NXB OTU N101:14/4 NXB OTU N101:14/5 NXB OTU N101:14/6 NXB OTU N101:14/7 NXB OTU N101:14/8 NXB OTU N101:14/9 NXB BST EQU L102:4 0 NXB EQU N103:4 0 BND ONS N101:5/4 MOV N101:14 N101:24 NXB EQU N101:14 0 BST CLR L102:4 NXB CLR N103:4 BND BND EOR
%   L102:4  "Biennial Maintenance Activity Cycles Remaining" %
%   N103:4  "Biennial Maintenance Activity Hours Remaining" %
%   N101:14  "Biennial Activity Enable" %
%   N101:24  "Biennial Activity Status" %

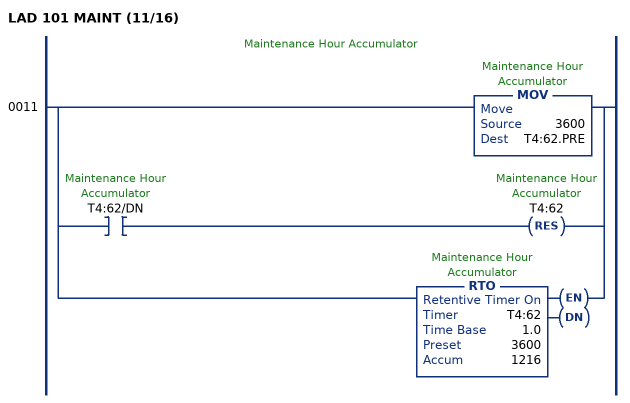
% Rung: 11 %
% Maintenance Hour Accumulator %
SOR BST MOV 3600 T4:62.PRE NXB XIC T4:62/DN RES T4:62 NXB RTO T4:62 1.0 3600 1216 BND EOR
%   T4:62  "Maintenance Hour Accumulator" %

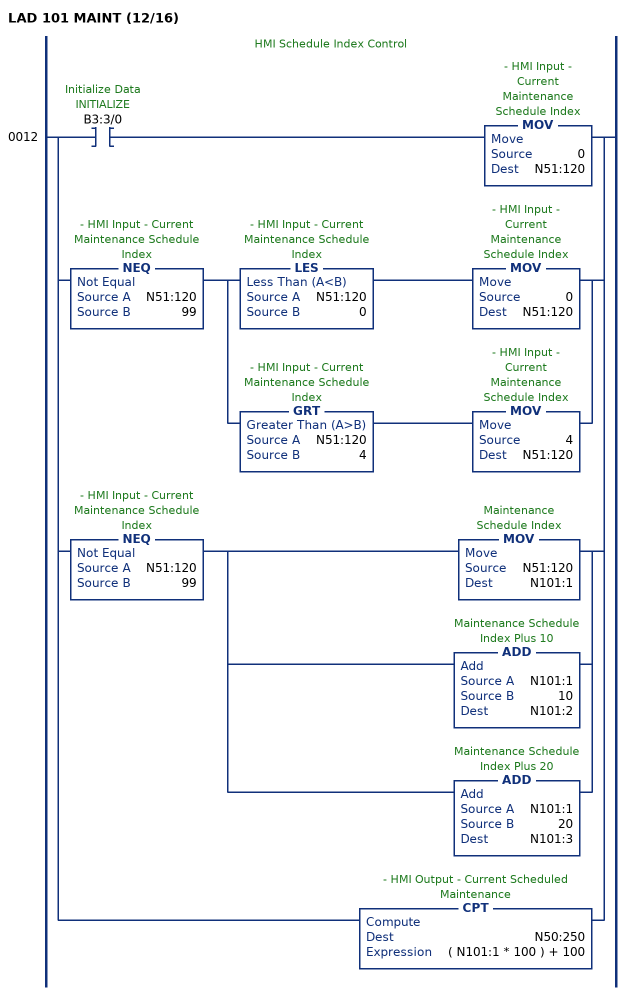
% Rung: 12 %
% HMI Schedule Index Control %
SOR BST BST XIC B3:3/0 MOV 0 N51:120 NXB NEQ N51:120 99 BST LES N51:120 0 MOV 0 N51:120 NXB GRT N51:120 4 MOV 4 N51:120 BND BND NXB NEQ N51:120 99 BST MOV N51:120 N101:1 NXB ADD N101:1 10 N101:2 NXB ADD N101:1 20 N101:3 BND NXB CPT N50:250 " ( N101:1 * 100 ) + 100 " BND EOR
%   B3:3/0  INITIALIZE  "Initialize Data" %
%   N51:120  "- HMI Input - Current Maintenance Schedule Index" %
%   N101:1  "Maintenance Schedule Index" %
%   N101:2  "Maintenance Schedule Index Plus 10" %
%   N101:3  "Maintenance Schedule Index Plus 20" %
%   N50:250  "- HMI Output - Current Scheduled Maintenance" %

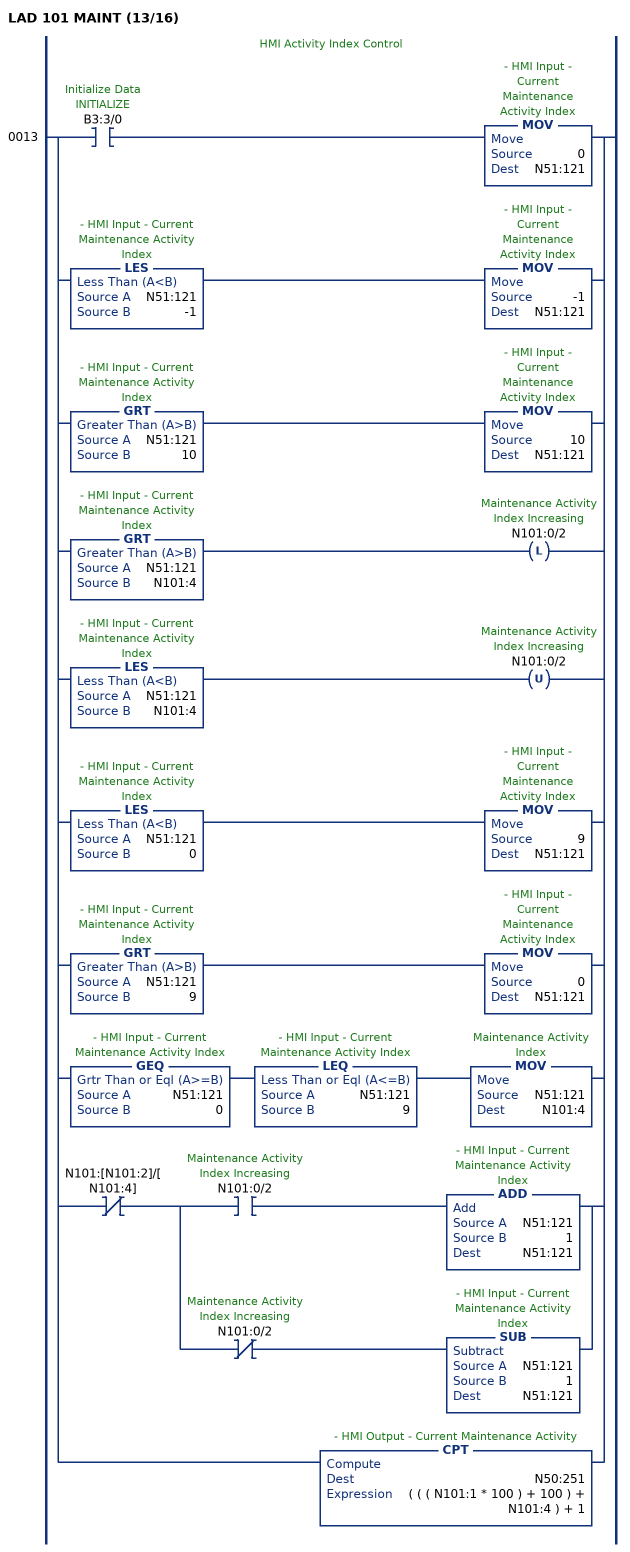
% Rung: 13 %
% HMI Activity Index Control %
SOR BST BST XIC B3:3/0 MOV 0 N51:121 NXB LES N51:121 -1 MOV -1 N51:121 NXB GRT N51:121 10 MOV 10 N51:121 BND NXB BST GRT N51:121 N101:4 OTL N101:0/2 NXB LES N51:121 N101:4 OTU N101:0/2 BND NXB BST LES N51:121 0 MOV 9 N51:121 NXB GRT N51:121 9 MOV 0 N51:121 NXB GEQ N51:121 0 LEQ N51:121 9 MOV N51:121 N101:4 BND NXB XIO N101:[N101:2]/[N101:4] BST XIC N101:0/2 ADD N51:121 1 N51:121 NXB XIO N101:0/2 SUB N51:121 1 N51:121 BND NXB CPT N50:251 " ( ( ( N101:1 * 100 ) + 100 ) + N101:4 ) + 1 " BND EOR
%   B3:3/0  INITIALIZE  "Initialize Data" %
%   N51:121  "- HMI Input - Current Maintenance Activity Index" %
%   N101:4  "Maintenance Activity Index" %
%   N101:0/2  "Maintenance Activity Index Increasing" %
%   N101:2  "Maintenance Schedule Index Plus 10" %
%   N50:251  "- HMI Output - Current Maintenance Activity" %
%   N101:1  "Maintenance Schedule Index" %

